TYPE OrderPLC :
STRUCT
	RobotPOS:STRING; //Prerequest position for the robot to do the step
	PLCorder:INT;	//PLCStep Code
	Robotreply:INT;	//Robot Response Code
END_STRUCT
END_TYPE

(* stored: Version 1.1.0.1, ProductVersion 3.1.4022.16
   DUT OrderPLC: Id {55b2a1cb-6b47-498f-b7ce-5c0304201352} *)
